// TIA Portal project "trafik_lamba_uygulama" (V14)

(* hardware
DEVICE "S71500/ET200MP station_1"  S7-1500 station
   slot 0: "Rail_0"  Rack  6ES7 590-1***0-0AA0
   slot 1: "PLC_1"  CPU 1511C-1 PN  6ES7 511-1CK00-0AB0  V2.0
      slot 3: "CPU display_1"  6ES7591-1AA00-0AA0
*)

// ===== PLC "PLC_1"  CPU 1511C-1 PN =====

VAR_GLOBAL   // PLC tag table "Default tag table"
   "start" AT %I0.1 : Bool;
   "yol_1-3" AT %Q0.0 : Bool;
   "yol_2-4" AT %Q0.1 : Bool;
   "kirmizi_isik_yol-1" AT %Q1.0 : Bool;
   "sari_isik_yol-1" AT %Q1.1 : Bool;
   "yesil_isik_yol-1" AT %Q1.2 : Bool;
   "reset" AT %I0.0 : Bool;
   "dongu" AT %M0.0 : Bool;
   "kirmizi_isik_yol-3" AT %Q1.3 : Bool;
   "sari_isik_yol-3" AT %Q1.4 : Bool;
   "yesil_isik_yol-3" AT %Q1.5 : Bool;
   "yol_5-6" AT %Q0.2 : Bool;
   "kirmizi_isik_yol-2" AT %Q2.0 : Bool;
   "sari_isik_yol-2" AT %Q2.1 : Bool;
   "yesil_isik_yol-2" AT %Q2.2 : Bool;
   "kirmizi_isik_yol-4" AT %Q2.3 : Bool;
   "sari_isik_yol-4" AT %Q2.4 : Bool;
   "yesil_isik_yol-4" AT %Q2.5 : Bool;
   "sistem" AT %Q10.0 : Bool;
   "yol_7-8" AT %Q0.3 : Bool;
   "kirmizi_isik_yol-5" AT %Q3.0 : Bool;
   "kirmizi_isik_yol-6" AT %Q3.3 : Bool;
   "sari_isik_yol-5" AT %Q3.1 : Bool;
   "sari_isik_yol-6" AT %Q3.4 : Bool;
   "yesil_isik_yol-5" AT %Q3.2 : Bool;
   "yesil_isik_yol-6" AT %Q3.5 : Bool;
   "kirmizi_isik_yol-7" AT %Q4.0 : Bool;
   "kirmizi_isik_yol-8" AT %Q4.3 : Bool;
   "sari_isik_yol-7" AT %Q4.1 : Bool;
   "sari_isik_yol-8" AT %Q4.4 : Bool;
   "yesil_isik_yol-7" AT %Q4.2 : Bool;
   "yesil_isik_yol-8" AT %Q4.5 : Bool;
END_VAR

// folder: System blocks/Program resources

DATA_BLOCK "zaman_yol_5-6"   // DB1
{ S7_Optimized_Access := 'TRUE' }
AUTHOR : Simatic
FAMILY : IEC
NAME : IEC_TMR
VERSION : 1.0
// stored: InstanceOfName IEC_TIMER
"IEC_TIMER"
BEGIN
END_DATA_BLOCK

DATA_BLOCK "zaman_yol_1-3"   // DB2
{ S7_Optimized_Access := 'TRUE' }
AUTHOR : Simatic
FAMILY : IEC
NAME : IEC_TMR
VERSION : 1.0
// stored: InstanceOfName IEC_TIMER
"IEC_TIMER"
BEGIN
END_DATA_BLOCK

DATA_BLOCK "zaman_yol_2-4"   // DB3
{ S7_Optimized_Access := 'TRUE' }
AUTHOR : Simatic
FAMILY : IEC
NAME : IEC_TMR
VERSION : 1.0
// stored: InstanceOfName IEC_TIMER
"IEC_TIMER"
BEGIN
END_DATA_BLOCK

DATA_BLOCK "zaman_yol_7-8"   // DB4
{ S7_Optimized_Access := 'TRUE' }
AUTHOR : Simatic
FAMILY : IEC
NAME : IEC_TMR
VERSION : 1.0
// stored: InstanceOfName IEC_TIMER
"IEC_TIMER"
BEGIN
END_DATA_BLOCK

// folder: (top level)

ORGANIZATION_BLOCK "Main"   // OB1, LAD, ProgramCycle
TITLE = "Main Program Sweep (Cycle)"
{ S7_Optimized_Access := 'TRUE' }
VERSION : 0.1
   VAR_INPUT
      Initial_Call : Bool;   // Initial call of this OB
      Remanence : Bool;   // =True, if remanent data are available
   END_VAR
   VAR_TEMP   // added for the SCL form of the ladder/FBD networks
      _w1 : Bool;
   END_VAR
BEGIN

REGION Network 1
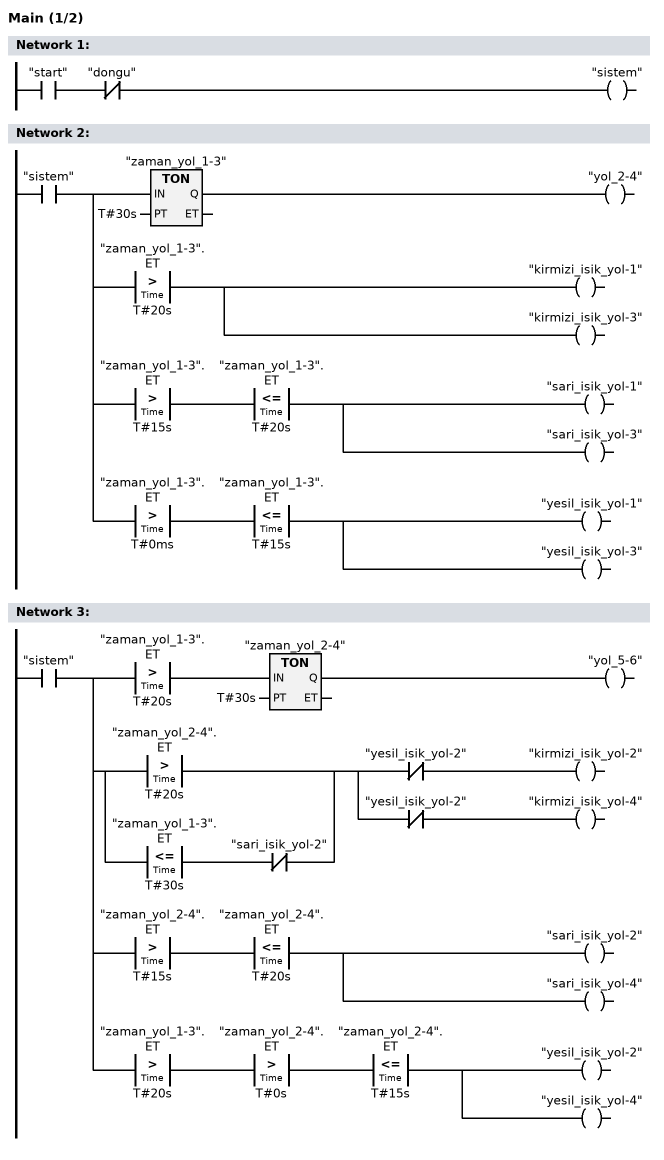
   RUNG wire#powerrail
      Contact( "start" )
      I_Contact( "dongu" )
      Coil( "sistem" )
   END_RUNG
   // the same network as SCL:
   "sistem" := "start" AND NOT "dongu";
END_REGION

REGION Network 2
   "zaman_yol_1-3".TON(IN := "sistem", PT := T#30s);
   "yol_2-4" := "zaman_yol_1-3".Q;
   "kirmizi_isik_yol-1" := "sistem" AND ("zaman_yol_1-3".ET > T#20s);
   "kirmizi_isik_yol-3" := "kirmizi_isik_yol-1";
   "sari_isik_yol-1" := "sistem" AND ("zaman_yol_1-3".ET > T#15s) AND ("zaman_yol_1-3".ET <= T#20s);
   "sari_isik_yol-3" := "sari_isik_yol-1";
   "yesil_isik_yol-1" := "sistem" AND ("zaman_yol_1-3".ET > T#0ms) AND ("zaman_yol_1-3".ET <= T#15s);
   "yesil_isik_yol-3" := "yesil_isik_yol-1";
END_REGION

REGION Network 3
   "zaman_yol_2-4".TON(IN := "sistem" AND ("zaman_yol_1-3".ET > T#20s), PT := T#30s);
   "yol_5-6" := "zaman_yol_2-4".Q;
   #_w1 := "sistem" AND (("zaman_yol_2-4".ET > T#20s) OR (("zaman_yol_1-3".ET <= T#30s) AND NOT "sari_isik_yol-2"));
   "kirmizi_isik_yol-2" := #_w1 AND NOT "yesil_isik_yol-2";
   "kirmizi_isik_yol-4" := #_w1 AND NOT "yesil_isik_yol-2";
   "sari_isik_yol-2" := "sistem" AND ("zaman_yol_2-4".ET > T#15s) AND ("zaman_yol_2-4".ET <= T#20s);
   "sari_isik_yol-4" := "sari_isik_yol-2";
   "yesil_isik_yol-2" := "sistem" AND ("zaman_yol_1-3".ET > T#20s) AND ("zaman_yol_2-4".ET > T#0s) AND ("zaman_yol_2-4".ET <= T#15s);
   "yesil_isik_yol-4" := "yesil_isik_yol-2";
END_REGION

REGION Network 4
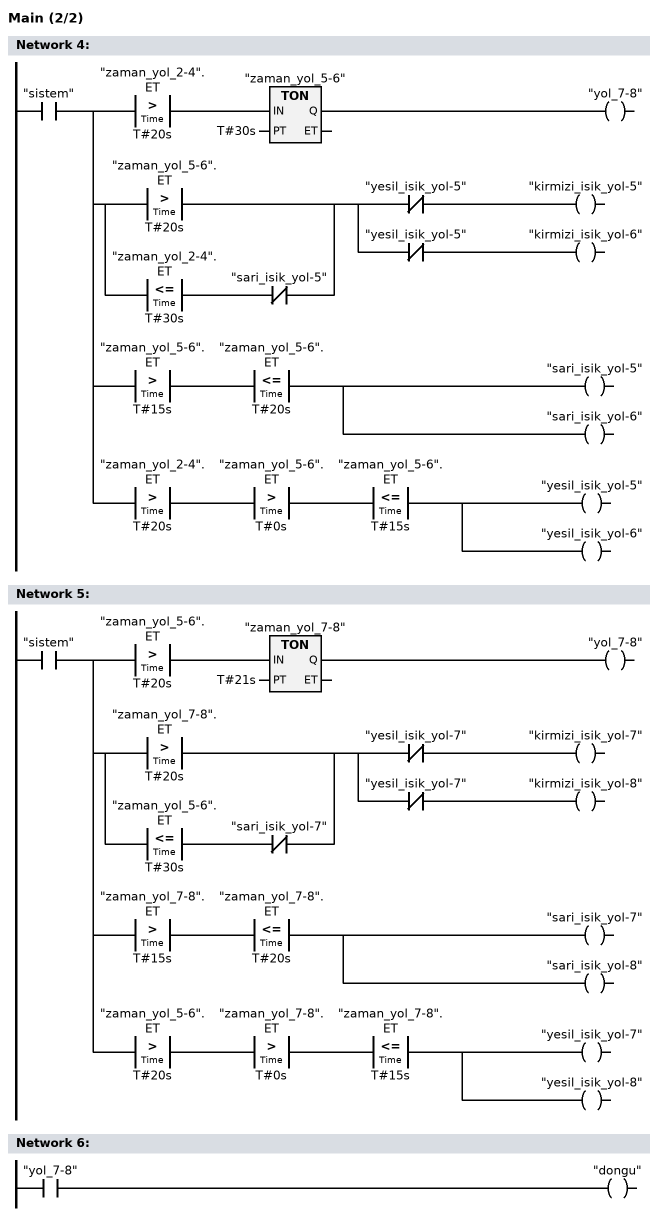
   "zaman_yol_5-6".TON(IN := "sistem" AND ("zaman_yol_2-4".ET > T#20s), PT := T#30s);
   "yol_7-8" := "zaman_yol_5-6".Q;
   #_w1 := "sistem" AND (("zaman_yol_5-6".ET > T#20s) OR (("zaman_yol_2-4".ET <= T#30s) AND NOT "sari_isik_yol-5"));
   "kirmizi_isik_yol-5" := #_w1 AND NOT "yesil_isik_yol-5";
   "kirmizi_isik_yol-6" := #_w1 AND NOT "yesil_isik_yol-5";
   "sari_isik_yol-5" := "sistem" AND ("zaman_yol_5-6".ET > T#15s) AND ("zaman_yol_5-6".ET <= T#20s);
   "sari_isik_yol-6" := "sari_isik_yol-5";
   "yesil_isik_yol-5" := "sistem" AND ("zaman_yol_2-4".ET > T#20s) AND ("zaman_yol_5-6".ET > T#0s) AND ("zaman_yol_5-6".ET <= T#15s);
   "yesil_isik_yol-6" := "yesil_isik_yol-5";
END_REGION

REGION Network 5
   "zaman_yol_7-8".TON(IN := "sistem" AND ("zaman_yol_5-6".ET > T#20s), PT := T#21s);
   "yol_7-8" := "zaman_yol_7-8".Q;
   #_w1 := "sistem" AND (("zaman_yol_7-8".ET > T#20s) OR (("zaman_yol_5-6".ET <= T#30s) AND NOT "sari_isik_yol-7"));
   "kirmizi_isik_yol-7" := #_w1 AND NOT "yesil_isik_yol-7";
   "kirmizi_isik_yol-8" := #_w1 AND NOT "yesil_isik_yol-7";
   "sari_isik_yol-7" := "sistem" AND ("zaman_yol_7-8".ET > T#15s) AND ("zaman_yol_7-8".ET <= T#20s);
   "sari_isik_yol-8" := "sari_isik_yol-7";
   "yesil_isik_yol-7" := "sistem" AND ("zaman_yol_5-6".ET > T#20s) AND ("zaman_yol_7-8".ET > T#0s) AND ("zaman_yol_7-8".ET <= T#15s);
   "yesil_isik_yol-8" := "yesil_isik_yol-7";
END_REGION

REGION Network 6
   RUNG wire#powerrail
      Contact( "yol_7-8" )
      Coil( "dongu" )
   END_RUNG
   // the same network as SCL:
   "dongu" := "yol_7-8";
END_REGION
END_ORGANIZATION_BLOCK